   1:  PR[91,2] = PR[90,2] + 14.295;
   1:L PR[91] R[100]mm/sec CNT100;
   1:  PR[91,1] = PR[90,1] + 9.800;
   1:  PR[91,2] = PR[90,2] + 14.166;
   1:L PR[91] R[100]mm/sec CNT100;
   1:  PR[91,1] = PR[90,1] + 6.679;
   1:  PR[91,2] = PR[90,2] + 10.931;
   1:L PR[91] R[100]mm/sec CNT100;
   1:  PR[91,1] = PR[90,1] + 6.224;
   1:  PR[91,2] = PR[90,2] + 10.258;
   1:L PR[91] R[100]mm/sec CNT100;
   1:  PR[91,1] = PR[90,1] + 5.273;
   1:  PR[91,2] = PR[90,2] + 8.564;
   1:L PR[91] R[100]mm/sec CNT100;
   1:  PR[91,1] = PR[90,1] + 5.411;
   1:  PR[91,2] = PR[90,2] + 8.540;
   1:L PR[91] R[100]mm/sec CNT100;
   1:  PR[91,1] = PR[90,1] + 3.886;
   1:  PR[91,2] = PR[90,2] + 6.154;
   1:L PR[91] R[100]mm/sec CNT100;
   1:  PR[91,1] = PR[90,1] + 3.596;
   1:  PR[91,2] = PR[90,2] + 5.846;
   1:L PR[91] R[100]mm/sec CNT100;
   1:  PR[91,1] = PR[90,1] + 2.742;
   1:  PR[91,2] = PR[90,2] + 5.238;
   1:L PR[91] R[100]mm/sec CNT100;
   1:  PR[91,1] = PR[90,1] + 1.672;
   1:  PR[91,2] = PR[90,2] + 5.008;
   1:L PR[91] R[100]mm/sec CNT100;
   1:  PR[91,1] = PR[90,1] + -1.507;
   1:L PR[91] R[100]mm/sec CNT100;
   1:  PR[91] = PR[90];
   1:  PR[91,1] = PR[90,1] + -2.515;
   1:  PR[91,2] = PR[90,2] + 5.532;
   1:  PR[91,3] = PR[90,3] + 14.945;
   1:L PR[91] R[100]mm/sec CNT100;
   1:  PR[91,1] = PR[90,1] + -3.313;
   1:  PR[91,2] = PR[90,2] + 6.100;
   1:L PR[91] R[100]mm/sec CNT100;
   1:  PR[91,1] = PR[90,1] + -3.690;
   1:  PR[91,2] = PR[90,2] + 6.481;
   1:L PR[91] R[100]mm/sec CNT100;
   1:  PR[91,1] = PR[90,1] + -4.029;
   1:  PR[91,2] = PR[90,2] + 7.015;
   1:L PR[91] R[100]mm/sec CNT100;
   1:  PR[91,1] = PR[90,1] + -5.541;
   1:  PR[91,2] = PR[90,2] + 9.725;
   1:L PR[91] R[100]mm/sec CNT100;
   1:  PR[91,1] = PR[90,1] + -6.491;
   1:  PR[91,2] = PR[90,2] + 11.148;
   1:L PR[91] R[100]mm/sec CNT100;
   1:  PR[91,1] = PR[90,1] + -9.060;
   1:  PR[91,2] = PR[90,2] + 13.805;
   1:L PR[91] R[100]mm/sec CNT100;
   1:  PR[91,1] = PR[90,1] + -9.776;
   1:  PR[91,2] = PR[90,2] + 14.440;
   1:L PR[91] R[100]mm/sec CNT100;
   1:  PR[91,1] = PR[90,1] + -13.611;
   1:  PR[91,2] = PR[90,2] + 16.788;
   1:L PR[91] R[100]mm/sec CNT100;
   1:  PR[91,1] = PR[90,1] + -13.803;
   1:  PR[91,2] = PR[90,2] + 16.888;
   1:L PR[91] R[100]mm/sec CNT100;
   1:  PR[91,1] = PR[90,1] + -16.097;
   1:  PR[91,2] = PR[90,2] + 17.603;
   1:L PR[91] R[100]mm/sec CNT100;
   1:  PR[91,1] = PR[90,1] + -18.417;
   1:  PR[91,2] = PR[90,2] + 18.357;
   1:L PR[91] R[100]mm/sec CNT100;
   1:  PR[91,1] = PR[90,1] + -18.598;
   1:  PR[91,2] = PR[90,2] + 18.378;
   1:L PR[91] R[100]mm/sec CNT100;
   1:  PR[91,1] = PR[90,1] + -23.160;
   1:  PR[91,2] = PR[90,2] + 18.675;
   1:L PR[91] R[100]mm/sec CNT100;
   1:  PR[91,1] = PR[90,1] + -24.014;
   1:  PR[91,2] = PR[90,2] + 18.553;
   1:L PR[91] R[100]mm/sec CNT100;
   1:  PR[91,1] = PR[90,1] + -27.876;
   1:  PR[91,2] = PR[90,2] + 17.835;
   1:L PR[91] R[100]mm/sec CNT100;
   1:  PR[91,1] = PR[90,1] + -29.208;
   1:  PR[91,2] = PR[90,2] + 17.272;
   1:L PR[91] R[100]mm/sec CNT100;
   1:  PR[91,1] = PR[90,1] + -32.267;
   1:  PR[91,2] = PR[90,2] + 15.857;
   1:L PR[91] R[100]mm/sec CNT100;
   1:  PR[91,1] = PR[90,1] + -33.781;
   1:  PR[91,2] = PR[90,2] + 14.686;
   1:L PR[91] R[100]mm/sec CNT100;
   1:  PR[91,1] = PR[90,1] + -36.042;
   1:  PR[91,2] = PR[90,2] + 12.845;
   1:L PR[91] R[100]mm/sec CNT100;
   1:  PR[91,1] = PR[90,1] + -37.414;
   1:  PR[91,2] = PR[90,2] + 11.050;
   1:L PR[91] R[100]mm/sec CNT100;
   1:  PR[91,1] = PR[90,1] + -38.944;
   1:  PR[91,2] = PR[90,2] + 8.967;
   1:L PR[91] R[100]mm/sec CNT100;
   1:  PR[91,1] = PR[90,1] + -39.896;
   1:  PR[91,2] = PR[90,2] + 6.669;
   1:L PR[91] R[100]mm/sec CNT100;
   1:  PR[91,1] = PR[90,1] + -40.771;
   1:  PR[91,2] = PR[90,2] + 4.501;
   1:L PR[91] R[100]mm/sec CNT100;
   1:  PR[91,1] = PR[90,1] + -41.398;
   1:  PR[91,2] = PR[90,2] + -0.312;
   1:L PR[91] R[100]mm/sec CNT100;
   1:  PR[91,1] = PR[90,1] + -40.771;
   1:  PR[91,2] = PR[90,2] + -5.125;
   1:L PR[91] R[100]mm/sec CNT100;
   1:  PR[91,1] = PR[90,1] + -39.896;
   1:  PR[91,2] = PR[90,2] + -7.294;
   1:L PR[91] R[100]mm/sec CNT100;
   1:  PR[91,1] = PR[90,1] + -38.944;
   1:  PR[91,2] = PR[90,2] + -9.591;
   1:L PR[91] R[100]mm/sec CNT100;
   1:  PR[91,1] = PR[90,1] + -37.414;
   1:  PR[91,2] = PR[90,2] + -11.674;
   1:L PR[91] R[100]mm/sec CNT100;
   1:  PR[91,1] = PR[90,1] + -36.042;
   1:  PR[91,2] = PR[90,2] + -13.469;
   1:L PR[91] R[100]mm/sec CNT100;
   1:  PR[91,1] = PR[90,1] + -33.781;
   1:  PR[91,2] = PR[90,2] + -15.310;
   1:L PR[91] R[100]mm/sec CNT100;
   1:  PR[91,1] = PR[90,1] + -32.266;
   1:  PR[91,2] = PR[90,2] + -16.481;
   1:L PR[91] R[100]mm/sec CNT100;
   1:  PR[91,1] = PR[90,1] + -29.208;
   1:  PR[91,2] = PR[90,2] + -17.896;
   1:L PR[91] R[100]mm/sec CNT100;
   1:  PR[91,1] = PR[90,1] + -27.875;
   1:  PR[91,2] = PR[90,2] + -18.459;
   1:L PR[91] R[100]mm/sec CNT100;
   1:  PR[91,1] = PR[90,1] + -24.013;
   1:  PR[91,2] = PR[90,2] + -19.177;
   1:L PR[91] R[100]mm/sec CNT100;
   1:  PR[91,1] = PR[90,1] + -23.159;
   1:  PR[91,2] = PR[90,2] + -19.299;
   1:L PR[91] R[100]mm/sec CNT100;
   1:  PR[91,1] = PR[90,1] + -18.596;
   1:  PR[91,2] = PR[90,2] + -19.001;
   1:L PR[91] R[100]mm/sec CNT100;
   1:  PR[91,1] = PR[90,1] + -18.416;
   1:  PR[91,2] = PR[90,2] + -18.981;
   1:L PR[91] R[100]mm/sec CNT100;
   1:  PR[91,1] = PR[90,1] + -16.097;
   1:  PR[91,2] = PR[90,2] + -18.227;
   1:L PR[91] R[100]mm/sec CNT100;
   1:  PR[91,1] = PR[90,1] + -13.802;
   1:  PR[91,2] = PR[90,2] + -17.512;
   1:L PR[91] R[100]mm/sec CNT100;
   1:  PR[91,1] = PR[90,1] + -13.610;
   1:  PR[91,2] = PR[90,2] + -17.411;
   1:L PR[91] R[100]mm/sec CNT100;
   1:  PR[91,1] = PR[90,1] + -9.775;
   1:  PR[91,2] = PR[90,2] + -15.063;
   1:L PR[91] R[100]mm/sec CNT100;
   1:  PR[91,1] = PR[90,1] + -9.059;
   1:  PR[91,2] = PR[90,2] + -14.428;
   1:L PR[91] R[100]mm/sec CNT100;
   1:  PR[91,1] = PR[90,1] + -6.489;
   1:  PR[91,2] = PR[90,2] + -11.769;
   1:L PR[91] R[100]mm/sec CNT100;
   1:  PR[91,1] = PR[90,1] + -5.569;
   1:  PR[91,2] = PR[90,2] + -10.401;
   1:L PR[91] R[100]mm/sec CNT100;
   1:  PR[91,1] = PR[90,1] + -4.028;
   1:  PR[91,2] = PR[90,2] + -7.639;
   1:L PR[91] R[100]mm/sec CNT100;
   1:  PR[91,1] = PR[90,1] + -3.683;
   1:  PR[91,2] = PR[90,2] + -7.096;
   1:L PR[91] R[100]mm/sec CNT100;
   1:  PR[91,1] = PR[90,1] + -3.311;
   1:  PR[91,2] = PR[90,2] + -6.722;
   1:L PR[91] R[100]mm/sec CNT100;
   1:  PR[91,1] = PR[90,1] + -2.515;
   1:  PR[91,2] = PR[90,2] + -6.156;
   1:L PR[91] R[100]mm/sec CNT100;
   1:  PR[91,1] = PR[90,1] + -1.428;
   1:  PR[91,2] = PR[90,2] + -5.921;
   1:L PR[91] R[100]mm/sec CNT100;
   1:  PR[91,1] = PR[90,1] + 1.584;
   1:L PR[91] R[100]mm/sec CNT100;
   1:  PR[91,1] = PR[90,1] + 2.668;
   1:  PR[91,2] = PR[90,2] + -6.155;
   1:L PR[91] R[100]mm/sec CNT100;
   1:  PR[91,1] = PR[90,1] + 3.441;
   1:  PR[91,2] = PR[90,2] + -6.703;
   1:L PR[91] R[100]mm/sec CNT100;
   1:  PR[91,1] = PR[90,1] + 3.541;
   1:  PR[91,2] = PR[90,2] + -6.796;
   1:L PR[91] R[100]mm/sec CNT100;
   1:  PR[91,1] = PR[90,1] + 3.696;
   1:  PR[91,2] = PR[90,2] + -6.767;
   1:L PR[91] R[100]mm/sec CNT100;
   1:  PR[91,1] = PR[90,1] + 5.726;
   1:  PR[91,2] = PR[90,2] + -10.398;
   1:L PR[91] R[100]mm/sec CNT100;
   1:  PR[91,1] = PR[90,1] + 6.644;
   1:  PR[91,2] = PR[90,2] + -11.761;
   1:L PR[91] R[100]mm/sec CNT100;
   1:  PR[91,1] = PR[90,1] + 9.214;
   1:  PR[91,2] = PR[90,2] + -14.427;
   1:L PR[91] R[100]mm/sec CNT100;
   1:  PR[91,1] = PR[90,1] + 9.930;
   1:  PR[91,2] = PR[90,2] + -15.063;
   1:L PR[91] R[100]mm/sec CNT100;
   1:  PR[91,1] = PR[90,1] + 13.762;
   1:  PR[91,2] = PR[90,2] + -17.409;
   1:L PR[91] R[100]mm/sec CNT100;
   1:  PR[91,1] = PR[90,1] + 13.954;
   1:  PR[91,2] = PR[90,2] + -17.510;
   1:L PR[91] R[100]mm/sec CNT100;
   1:  PR[91,1] = PR[90,1] + 16.254;
   1:  PR[91,2] = PR[90,2] + -18.227;
   1:L PR[91] R[100]mm/sec CNT100;
   1:  PR[91,1] = PR[90,1] + 18.569;
   1:  PR[91,2] = PR[90,2] + -18.980;
   1:L PR[91] R[100]mm/sec CNT100;
   1:  PR[91,1] = PR[90,1] + 18.749;
   1:  PR[91,2] = PR[90,2] + -19.001;
   1:L PR[91] R[100]mm/sec CNT100;
   1:  PR[91,1] = PR[90,1] + 23.313;
   1:  PR[91,2] = PR[90,2] + -19.299;
   1:L PR[91] R[100]mm/sec CNT100;
   1:  PR[91,1] = PR[90,1] + 24.167;
   1:  PR[91,2] = PR[90,2] + -19.177;
   1:L PR[91] R[100]mm/sec CNT100;
   1:  PR[91,1] = PR[90,1] + 28.030;
   1:  PR[91,2] = PR[90,2] + -18.459;
   1:L PR[91] R[100]mm/sec CNT100;
   1:  PR[91,1] = PR[90,1] + 29.362;
   1:  PR[91,2] = PR[90,2] + -17.896;
   1:L PR[91] R[100]mm/sec CNT100;
   1:  PR[91,1] = PR[90,1] + 32.422;
   1:  PR[91,2] = PR[90,2] + -16.482;
   1:L PR[91] R[100]mm/sec CNT100;
   1:  PR[91,1] = PR[90,1] + 33.936;
   1:  PR[91,2] = PR[90,2] + -15.312;
   1:L PR[91] R[100]mm/sec CNT100;
   1:  PR[91,1] = PR[90,1] + 36.198;
   1:  PR[91,2] = PR[90,2] + -13.470;
   1:L PR[91] R[100]mm/sec CNT100;
   1:  PR[91,1] = PR[90,1] + 37.570;
   1:  PR[91,2] = PR[90,2] + -11.674;
   1:L PR[91] R[100]mm/sec CNT100;
   1:  PR[91,1] = PR[90,1] + 39.100;
   1:  PR[91,2] = PR[90,2] + -9.588;
   1:L PR[91] R[100]mm/sec CNT100;
   1:  PR[91,1] = PR[90,1] + 40.053;
   1:  PR[91,2] = PR[90,2] + -7.294;
   1:L PR[91] R[100]mm/sec CNT100;
   1:  PR[91,1] = PR[90,1] + 40.929;
   1:  PR[91,2] = PR[90,2] + -5.130;
   1:L PR[91] R[100]mm/sec CNT100;
   1:  PR[91,1] = PR[90,1] + 41.281;
   1:  PR[91,2] = PR[90,2] + -2.473;
   1:L PR[91] R[100]mm/sec CNT100;
   1:  PR[91,1] = PR[90,1] + 41.555;
   1:  PR[91,2] = PR[90,2] + -0.314;
   1:L PR[91] R[100]mm/sec CNT100;
   1:  PR[91,1] = PR[90,1] + 40.928;
   1:  PR[91,2] = PR[90,2] + 4.508;
   1:L PR[91] R[100]mm/sec CNT100;
   1:  PR[91,1] = PR[90,1] + 40.053;
   1:  PR[91,2] = PR[90,2] + 6.669;
   1:L PR[91] R[100]mm/sec CNT100;
   1:  PR[91,1] = PR[90,1] + 39.100;
   1:  PR[91,2] = PR[90,2] + 8.965;
   1:L PR[91] R[100]mm/sec CNT100;
   1:  PR[91,1] = PR[90,1] + 37.570;
   1:  PR[91,2] = PR[90,2] + 11.050;
   1:L PR[91] R[100]mm/sec CNT100;
   1:  PR[91,1] = PR[90,1] + 36.198;
   1:  PR[91,2] = PR[90,2] + 12.846;
   1:L PR[91] R[100]mm/sec CNT100;
   1:  PR[91,1] = PR[90,1] + 33.937;
   1:  PR[91,2] = PR[90,2] + 14.688;
   1:L PR[91] R[100]mm/sec CNT100;
   1:  PR[91,1] = PR[90,1] + 32.422;
   1:  PR[91,2] = PR[90,2] + 15.858;
   1:L PR[91] R[100]mm/sec CNT100;
   1:  PR[91,1] = PR[90,1] + 29.364;
   1:  PR[91,2] = PR[90,2] + 17.271;
   1:L PR[91] R[100]mm/sec CNT100;
   1:  PR[91,1] = PR[90,1] + 28.031;
   1:  PR[91,2] = PR[90,2] + 17.834;
   1:L PR[91] R[100]mm/sec CNT100;
   1:  PR[91,1] = PR[90,1] + 24.170;
   1:  PR[91,2] = PR[90,2] + 18.553;
   1:L PR[91] R[100]mm/sec CNT100;
   1:  PR[91,1] = PR[90,1] + 23.316;
   1:  PR[91,2] = PR[90,2] + 18.675;
   1:L PR[91] R[100]mm/sec CNT100;
   1:  PR[91,1] = PR[90,1] + 18.755;
   1:  PR[91,2] = PR[90,2] + 18.378;
   1:L PR[91] R[100]mm/sec CNT100;
   1:  PR[91,1] = PR[90,1] + 18.574;
   1:  PR[91,2] = PR[90,2] + 18.357;
   1:L PR[91] R[100]mm/sec CNT100;
   1:  PR[91,1] = PR[90,1] + 16.254;
   1:  PR[91,2] = PR[90,2] + 17.603;
   1:L PR[91] R[100]mm/sec CNT100;
   1:  PR[91,1] = PR[90,1] + 13.959;
   1:  PR[91,2] = PR[90,2] + 16.888;
   1:L PR[91] R[100]mm/sec CNT100;
   1:  PR[91,1] = PR[90,1] + 13.767;
   1:  PR[91,2] = PR[90,2] + 16.787;
   1:L PR[91] R[100]mm/sec CNT100;
   1:  PR[91,1] = PR[90,1] + 9.932;
   1:  PR[91,2] = PR[90,2] + 14.441;
   1:L PR[91] R[100]mm/sec CNT100;
   1:  PR[91,1] = PR[90,1] + 9.216;
   1:  PR[91,2] = PR[90,2] + 13.804;
   1:L PR[91] R[100]mm/sec CNT100;
   1:  PR[91,1] = PR[90,1] + 6.643;
   1:  PR[91,2] = PR[90,2] + 11.137;
   1:L PR[91] R[100]mm/sec CNT100;
   1:  PR[91,1] = PR[90,1] + 5.747;
   1:  PR[91,2] = PR[90,2] + 9.811;
   1:L PR[91] R[100]mm/sec CNT100;
   1:  PR[91,1] = PR[90,1] + 5.190;
   1:  PR[91,2] = PR[90,2] + 8.819;
   1:L PR[91] R[100]mm/sec CNT100;
   1:  PR[91,1] = PR[90,1] + 5.359;
   1:  PR[91,2] = PR[90,2] + 8.789;
   1:L PR[91] R[100]mm/sec CNT100;
   1:  PR[91,1] = PR[90,1] + 3.825;
   1:  PR[91,2] = PR[90,2] + 6.457;
   1:L PR[91] R[100]mm/sec CNT100;
   1:  PR[91,1] = PR[90,1] + 3.465;
   1:  PR[91,2] = PR[90,2] + 6.097;
   1:L PR[91] R[100]mm/sec CNT100;
   1:  PR[91,1] = PR[90,1] + 2.673;
   1:  PR[91,2] = PR[90,2] + 5.533;
   1:L PR[91] R[100]mm/sec CNT100;
   1:  PR[91,1] = PR[90,1] + 1.593;
   1:  PR[91,2] = PR[90,2] + 5.297;
   1:L PR[91] R[100]mm/sec CNT100;
   1:  PR[91,1] = PR[90,1] + -1.427;
   1:L PR[91] R[100]mm/sec CNT100;
   1:  PR[91] = PR[90];
   1:  PR[91,1] = PR[90,1] + -2.445;
   1:  PR[91,2] = PR[90,2] + 5.827;
   1:  PR[91,3] = PR[90,3] + 15.555;
   1:L PR[91] R[100]mm/sec CNT100;
   1:  PR[91,1] = PR[90,1] + -3.200;
   1:  PR[91,2] = PR[90,2] + 6.364;
   1:L PR[91] R[100]mm/sec CNT100;
   1:  PR[91,1] = PR[90,1] + -3.672;
   1:  PR[91,2] = PR[90,2] + 6.843;
   1:L PR[91] R[100]mm/sec CNT100;
   1:  PR[91,1] = PR[90,1] + -3.947;
   1:  PR[91,2] = PR[90,2] + 7.275;
   1:L PR[91] R[100]mm/sec CNT100;
   1:  PR[91,1] = PR[90,1] + -5.042;
   1:  PR[91,2] = PR[90,2] + 9.237;
   1:L PR[91] R[100]mm/sec CNT100;
   1:  PR[91,1] = PR[90,1] + -6.455;
   1:  PR[91,2] = PR[90,2] + 11.355;
   1:L PR[91] R[100]mm/sec CNT100;
   1:  PR[91,1] = PR[90,1] + -8.477;
   1:  PR[91,2] = PR[90,2] + 13.446;
   1:L PR[91] R[100]mm/sec CNT100;
   1:  PR[91,1] = PR[90,1] + -9.764;
   1:  PR[91,2] = PR[90,2] + 14.587;
   1:L PR[91] R[100]mm/sec CNT100;
   1:  PR[91,1] = PR[90,1] + -12.951;
   1:  PR[91,2] = PR[90,2] + 16.538;
   1:L PR[91] R[100]mm/sec CNT100;
   1:  PR[91,1] = PR[90,1] + -13.796;
   1:  PR[91,2] = PR[90,2] + 16.982;
   1:L PR[91] R[100]mm/sec CNT100;
   1:  PR[91,1] = PR[90,1] + -18.202;
   1:  PR[91,2] = PR[90,2] + 18.354;
   1:L PR[91] R[100]mm/sec CNT100;
   1:  PR[91,1] = PR[90,1] + -18.339;
   1:  PR[91,2] = PR[90,2] + 18.388;
   1:L PR[91] R[100]mm/sec CNT100;
   1:  PR[91,1] = PR[90,1] + -20.244;
   1:  PR[91,2] = PR[90,2] + 18.495;
   1:L PR[91] R[100]mm/sec CNT100;
   1:  PR[91,1] = PR[90,1] + -23.180;
   1:  PR[91,2] = PR[90,2] + 18.687;
   1:L PR[91] R[100]mm/sec CNT100;
   1:  PR[91,1] = PR[90,1] + -23.424;
   1:  PR[91,2] = PR[90,2] + 18.652;
   1:L PR[91] R[100]mm/sec CNT100;
   1:  PR[91,1] = PR[90,1] + -27.877;
   1:  PR[91,2] = PR[90,2] + 17.824;
   1:L PR[91] R[100]mm/sec CNT100;
   1:  PR[91,1] = PR[90,1] + -28.676;
   1:  PR[91,2] = PR[90,2] + 17.486;
   1:L PR[91] R[100]mm/sec CNT100;
   1:  PR[91,1] = PR[90,1] + -32.247;
   1:  PR[91,2] = PR[90,2] + 15.834;
   1:L PR[91] R[100]mm/sec CNT100;
   1:  PR[91,1] = PR[90,1] + -33.331;
   1:  PR[91,2] = PR[90,2] + 14.997;
   1:L PR[91] R[100]mm/sec CNT100;
   1:  PR[91,1] = PR[90,1] + -36.004;
   1:  PR[91,2] = PR[90,2] + 12.821;
   1:L PR[91] R[100]mm/sec CNT100;
   1:  PR[91,1] = PR[90,1] + -37.062;
   1:  PR[91,2] = PR[90,2] + 11.436;
   1:L PR[91] R[100]mm/sec CNT100;
   1:  PR[91,1] = PR[90,1] + -38.891;
   1:  PR[91,2] = PR[90,2] + 8.946;
   1:L PR[91] R[100]mm/sec CNT100;
   1:  PR[91,1] = PR[90,1] + -39.654;
   1:  PR[91,2] = PR[90,2] + 7.105;
   1:L PR[91] R[100]mm/sec CNT100;
   1:  PR[91,1] = PR[90,1] + -40.709;
   1:  PR[91,2] = PR[90,2] + 4.492;
   1:L PR[91] R[100]mm/sec CNT100;
   1:  PR[91,1] = PR[90,1] + -41.332;
   1:  PR[91,2] = PR[90,2] + -0.312;
   1:L PR[91] R[100]mm/sec CNT100;
   1:  PR[91,1] = PR[90,1] + -40.709;
   1:  PR[91,2] = PR[90,2] + -5.116;
   1:L PR[91] R[100]mm/sec CNT100;
   1:  PR[91,1] = PR[90,1] + -39.653;
   1:  PR[91,2] = PR[90,2] + -7.730;
   1:L PR[91] R[100]mm/sec CNT100;
   1:  PR[91,1] = PR[90,1] + -38.891;
   1:  PR[91,2] = PR[90,2] + -9.570;
   1:L PR[91] R[100]mm/sec CNT100;
   1:  PR[91,1] = PR[90,1] + -37.062;
   1:  PR[91,2] = PR[90,2] + -12.060;
   1:L PR[91] R[100]mm/sec CNT100;
   1:  PR[91,1] = PR[90,1] + -36.003;
   1:  PR[91,2] = PR[90,2] + -13.445;
   1:L PR[91] R[100]mm/sec CNT100;
   1:  PR[91,1] = PR[90,1] + -33.330;
   1:  PR[91,2] = PR[90,2] + -15.621;
   1:L PR[91] R[100]mm/sec CNT100;
   1:  PR[91,1] = PR[90,1] + -32.247;
   1:  PR[91,2] = PR[90,2] + -16.459;
   1:L PR[91] R[100]mm/sec CNT100;
   1:  PR[91,1] = PR[90,1] + -28.676;
   1:  PR[91,2] = PR[90,2] + -18.111;
   1:L PR[91] R[100]mm/sec CNT100;
   1:  PR[91,1] = PR[90,1] + -27.876;
   1:  PR[91,2] = PR[90,2] + -18.449;
   1:L PR[91] R[100]mm/sec CNT100;
   1:  PR[91,1] = PR[90,1] + -23.422;
   1:  PR[91,2] = PR[90,2] + -19.276;
   1:L PR[91] R[100]mm/sec CNT100;
   1:  PR[91,1] = PR[90,1] + -23.180;
   1:  PR[91,2] = PR[90,2] + -19.311;
   1:L PR[91] R[100]mm/sec CNT100;
   1:  PR[91,1] = PR[90,1] + -20.244;
   1:  PR[91,2] = PR[90,2] + -19.119;
   1:L PR[91] R[100]mm/sec CNT100;
   1:  PR[91,1] = PR[90,1] + -18.338;
   1:  PR[91,2] = PR[90,2] + -19.012;
   1:L PR[91] R[100]mm/sec CNT100;
   1:  PR[91,1] = PR[90,1] + -18.201;
   1:  PR[91,2] = PR[90,2] + -18.978;
   1:L PR[91] R[100]mm/sec CNT100;
   1:  PR[91,1] = PR[90,1] + -13.795;
   1:  PR[91,2] = PR[90,2] + -17.606;
   1:L PR[91] R[100]mm/sec CNT100;
   1:  PR[91,1] = PR[90,1] + -12.950;
   1:  PR[91,2] = PR[90,2] + -17.162;
   1:L PR[91] R[100]mm/sec CNT100;
   1:  PR[91,1] = PR[90,1] + -9.763;
   1:  PR[91,2] = PR[90,2] + -15.210;
   1:L PR[91] R[100]mm/sec CNT100;
   1:  PR[91,1] = PR[90,1] + -8.476;
   1:  PR[91,2] = PR[90,2] + -14.069;
   1:L PR[91] R[100]mm/sec CNT100;
   1:  PR[91,1] = PR[90,1] + -6.453;
   1:  PR[91,2] = PR[90,2] + -11.977;
   1:L PR[91] R[100]mm/sec CNT100;
   1:  PR[91,1] = PR[90,1] + -5.082;
   1:  PR[91,2] = PR[90,2] + -9.937;
   1:L PR[91] R[100]mm/sec CNT100;
   1:  PR[91,1] = PR[90,1] + -3.945;
   1:  PR[91,2] = PR[90,2] + -7.899;
   1:L PR[91] R[100]mm/sec CNT100;
   1:  PR[91,1] = PR[90,1] + -3.663;
   1:  PR[91,2] = PR[90,2] + -7.454;
   1:L PR[91] R[100]mm/sec CNT100;
   1:  PR[91,1] = PR[90,1] + -3.197;
   1:  PR[91,2] = PR[90,2] + -6.986;
   1:L PR[91] R[100]mm/sec CNT100;
   1:  PR[91,1] = PR[90,1] + -2.445;
   1:  PR[91,2] = PR[90,2] + -6.451;
   1:L PR[91] R[100]mm/sec CNT100;
   1:  PR[91,1] = PR[90,1] + -1.349;
   1:  PR[91,2] = PR[90,2] + -6.209;
   1:L PR[91] R[100]mm/sec CNT100;
   1:  PR[91,1] = PR[90,1] + 1.505;
   1:L PR[91] R[100]mm/sec CNT100;
   1:  PR[91,1] = PR[90,1] + 2.599;
   1:  PR[91,2] = PR[90,2] + -6.450;
   1:L PR[91] R[100]mm/sec CNT100;
   1:  PR[91,1] = PR[90,1] + 3.328;
   1:  PR[91,2] = PR[90,2] + -6.967;
   1:L PR[91] R[100]mm/sec CNT100;
   1:  PR[91,1] = PR[90,1] + 3.430;
   1:  PR[91,2] = PR[90,2] + -7.062;
   1:L PR[91] R[100]mm/sec CNT100;
   1:  PR[91,1] = PR[90,1] + 3.614;
   1:  PR[91,2] = PR[90,2] + -7.027;
   1:L PR[91] R[100]mm/sec CNT100;
   1:  PR[91,1] = PR[90,1] + 5.241;
   1:  PR[91,2] = PR[90,2] + -9.937;
   1:L PR[91] R[100]mm/sec CNT100;
   1:  PR[91,1] = PR[90,1] + 6.608;
   1:  PR[91,2] = PR[90,2] + -11.969;
   1:L PR[91] R[100]mm/sec CNT100;
   1:  PR[91,1] = PR[90,1] + 8.632;
   1:  PR[91,2] = PR[90,2] + -14.068;
   1:L PR[91] R[100]mm/sec CNT100;
   1:  PR[91,1] = PR[90,1] + 9.918;
   1:  PR[91,2] = PR[90,2] + -15.211;
   1:L PR[91] R[100]mm/sec CNT100;
   1:  PR[91,1] = PR[90,1] + 13.103;
   1:  PR[91,2] = PR[90,2] + -17.160;
   1:L PR[91] R[100]mm/sec CNT100;
   1:  PR[91,1] = PR[90,1] + 13.948;
   1:  PR[91,2] = PR[90,2] + -17.604;
   1:L PR[91] R[100]mm/sec CNT100;
   1:  PR[91,1] = PR[90,1] + 18.354;
   1:  PR[91,2] = PR[90,2] + -18.977;
   1:L PR[91] R[100]mm/sec CNT100;
   1:  PR[91,1] = PR[90,1] + 18.492;
   1:  PR[91,2] = PR[90,2] + -19.011;
   1:L PR[91] R[100]mm/sec CNT100;
   1:  PR[91,1] = PR[90,1] + 20.401;
   1:  PR[91,2] = PR[90,2] + -19.119;
   1:L PR[91] R[100]mm/sec CNT100;
   1:  PR[91,1] = PR[90,1] + 23.334;
   1:  PR[91,2] = PR[90,2] + -19.311;
   1:L PR[91] R[100]mm/sec CNT100;
   1:  PR[91,1] = PR[90,1] + 23.576;
   1:  PR[91,2] = PR[90,2] + -19.276;
   1:L PR[91] R[100]mm/sec CNT100;
   1:  PR[91,1] = PR[90,1] + 28.031;
   1:  PR[91,2] = PR[90,2] + -18.448;
   1:L PR[91] R[100]mm/sec CNT100;
   1:  PR[91,1] = PR[90,1] + 28.830;
   1:  PR[91,2] = PR[90,2] + -18.110;
   1:L PR[91] R[100]mm/sec CNT100;
   1:  PR[91,1] = PR[90,1] + 32.402;
   1:  PR[91,2] = PR[90,2] + -16.460;
   1:L PR[91] R[100]mm/sec CNT100;
   1:  PR[91,1] = PR[90,1] + 33.485;
   1:  PR[91,2] = PR[90,2] + -15.623;
   1:L PR[91] R[100]mm/sec CNT100;
   1:  PR[91,1] = PR[90,1] + 36.159;
   1:  PR[91,2] = PR[90,2] + -13.446;
   1:L PR[91] R[100]mm/sec CNT100;
   1:  PR[91,1] = PR[90,1] + 37.217;
   1:  PR[91,2] = PR[90,2] + -12.061;
   1:L PR[91] R[100]mm/sec CNT100;
   1:  PR[91,1] = PR[90,1] + 39.047;
   1:  PR[91,2] = PR[90,2] + -9.567;
   1:L PR[91] R[100]mm/sec CNT100;
   1:  PR[91,1] = PR[90,1] + 39.810;
   1:  PR[91,2] = PR[90,2] + -7.728;
   1:L PR[91] R[100]mm/sec CNT100;
   1:  PR[91,1] = PR[90,1] + 40.866;
   1:  PR[91,2] = PR[90,2] + -5.121;
   1:L PR[91] R[100]mm/sec CNT100;
   1:  PR[91,1] = PR[90,1] + 41.154;
   1:  PR[91,2] = PR[90,2] + -2.953;
   1:L PR[91] R[100]mm/sec CNT100;
   1:  PR[91,1] = PR[90,1] + 41.489;
   1:  PR[91,2] = PR[90,2] + -0.314;
   1:L PR[91] R[100]mm/sec CNT100;
   1:  PR[91,1] = PR[90,1] + 40.865;
   1:  PR[91,2] = PR[90,2] + 4.499;
   1:L PR[91] R[100]mm/sec CNT100;
   1:  PR[91,1] = PR[90,1] + 39.811;
   1:  PR[91,2] = PR[90,2] + 7.103;
   1:L PR[91] R[100]mm/sec CNT100;
   1:  PR[91,1] = PR[90,1] + 39.047;
   1:  PR[91,2] = PR[90,2] + 8.943;
   1:L PR[91] R[100]mm/sec CNT100;
   1:  PR[91,1] = PR[90,1] + 37.218;
   1:  PR[91,2] = PR[90,2] + 11.436;
   1:L PR[91] R[100]mm/sec CNT100;
   1:  PR[91,1] = PR[90,1] + 36.159;
   1:  PR[91,2] = PR[90,2] + 12.821;
   1:L PR[91] R[100]mm/sec CNT100;
   1:  PR[91,1] = PR[90,1] + 33.487;
   1:  PR[91,2] = PR[90,2] + 14.999;
   1:L PR[91] R[100]mm/sec CNT100;
   1:  PR[91,1] = PR[90,1] + 32.403;
   1:  PR[91,2] = PR[90,2] + 15.836;
   1:L PR[91] R[100]mm/sec CNT100;
   1:  PR[91,1] = PR[90,1] + 28.833;
   1:  PR[91,2] = PR[90,2] + 17.486;
   1:L PR[91] R[100]mm/sec CNT100;
   1:  PR[91,1] = PR[90,1] + 28.032;
   1:  PR[91,2] = PR[90,2] + 17.824;
   1:L PR[91] R[100]mm/sec CNT100;
   1:  PR[91,1] = PR[90,1] + 23.580;
   1:  PR[91,2] = PR[90,2] + 18.652;
   1:L PR[91] R[100]mm/sec CNT100;
   1:  PR[91,1] = PR[90,1] + 23.337;
   1:  PR[91,2] = PR[90,2] + 18.687;
   1:L PR[91] R[100]mm/sec CNT100;
   1:  PR[91,1] = PR[90,1] + 20.401;
   1:  PR[91,2] = PR[90,2] + 18.495;
   1:L PR[91] R[100]mm/sec CNT100;
   1:  PR[91,1] = PR[90,1] + 18.497;
   1:  PR[91,2] = PR[90,2] + 18.388;
   1:L PR[91] R[100]mm/sec CNT100;
   1:  PR[91,1] = PR[90,1] + 18.359;
   1:  PR[91,2] = PR[90,2] + 18.354;
   1:L PR[91] R[100]mm/sec CNT100;
   1:  PR[91,1] = PR[90,1] + 13.951;
   1:  PR[91,2] = PR[90,2] + 16.981;
   1:L PR[91] R[100]mm/sec CNT100;
   1:  PR[91,1] = PR[90,1] + 13.105;
   1:  PR[91,2] = PR[90,2] + 16.537;
   1:L PR[91] R[100]mm/sec CNT100;
   1:  PR[91,1] = PR[90,1] + 9.918;
   1:  PR[91,2] = PR[90,2] + 14.588;
   1:L PR[91] R[100]mm/sec CNT100;
   1:  PR[91,1] = PR[90,1] + 8.631;
   1:  PR[91,2] = PR[90,2] + 13.442;
   1:L PR[91] R[100]mm/sec CNT100;
   1:  PR[91,1] = PR[90,1] + 6.606;
   1:  PR[91,2] = PR[90,2] + 11.343;
   1:L PR[91] R[100]mm/sec CNT100;
   1:  PR[91,1] = PR[90,1] + 5.270;
   1:  PR[91,2] = PR[90,2] + 9.365;
   1:L PR[91] R[100]mm/sec CNT100;
   1:  PR[91,1] = PR[90,1] + 5.107;
   1:  PR[91,2] = PR[90,2] + 9.076;
   1:L PR[91] R[100]mm/sec CNT100;
   1:  PR[91,1] = PR[90,1] + 5.248;
   1:  PR[91,2] = PR[90,2] + 9.051;
   1:L PR[91] R[100]mm/sec CNT100;
   1:  PR[91,1] = PR[90,1] + 3.904;
   1:  PR[91,2] = PR[90,2] + 6.949;
   1:L PR[91] R[100]mm/sec CNT100;
   1:  PR[91,1] = PR[90,1] + 3.586;
   1:  PR[91,2] = PR[90,2] + 6.582;
   1:L PR[91] R[100]mm/sec CNT100;
   1:  PR[91,1] = PR[90,1] + 3.331;
   1:  PR[91,2] = PR[90,2] + 6.346;
   1:L PR[91] R[100]mm/sec CNT100;
   1:  PR[91,1] = PR[90,1] + 2.603;
   1:  PR[91,2] = PR[90,2] + 5.828;
   1:L PR[91] R[100]mm/sec CNT100;
   1:  PR[91,1] = PR[90,1] + 1.513;
   1:  PR[91,2] = PR[90,2] + 5.585;
   1:L PR[91] R[100]mm/sec CNT100;
   1:  PR[91,1] = PR[90,1] + -1.348;
   1:L PR[91] R[100]mm/sec CNT100;
   1:  PR[91] = PR[90];
   1:  PR[91,1] = PR[90,1] + -2.375;
   1:  PR[91,2] = PR[90,2] + 6.122;
   1:  PR[91,3] = PR[90,3] + 16.165;
   1:L PR[91] R[100]mm/sec CNT100;
   1:  PR[91,1] = PR[90,1] + -3.061;
   1:  PR[91,2] = PR[90,2] + 6.611;
   1:L PR[91] R[100]mm/sec CNT100;
   1:  PR[91,1] = PR[90,1] + -3.346;
   1:  PR[91,2] = PR[90,2] + 6.876;
   1:L PR[91] R[100]mm/sec CNT100;
   1:  PR[91,1] = PR[90,1] + -3.693;
   1:  PR[91,2] = PR[90,2] + 7.253;
   1:L PR[91] R[100]mm/sec CNT100;
   1:  PR[91,1] = PR[90,1] + -4.539;
   1:  PR[91,2] = PR[90,2] + 8.744;
   1:L PR[91] R[100]mm/sec CNT100;
   1:  PR[91,1] = PR[90,1] + -6.420;
   1:  PR[91,2] = PR[90,2] + 11.562;
   1:L PR[91] R[100]mm/sec CNT100;
   1:  PR[91,1] = PR[90,1] + -7.895;
   1:  PR[91,2] = PR[90,2] + 13.088;
   1:L PR[91] R[100]mm/sec CNT100;
   1:  PR[91,1] = PR[90,1] + -9.752;
   1:  PR[91,2] = PR[90,2] + 14.734;
   1:L PR[91] R[100]mm/sec CNT100;
   1:  PR[91,1] = PR[90,1] + -12.291;
   1:  PR[91,2] = PR[90,2] + 16.289;
   1:L PR[91] R[100]mm/sec CNT100;
   1:  PR[91,1] = PR[90,1] + -13.790;
   1:  PR[91,2] = PR[90,2] + 17.076;
   1:L PR[91] R[100]mm/sec CNT100;
   1:  PR[91,1] = PR[90,1] + -17.504;
   1:  PR[91,2] = PR[90,2] + 18.232;
   1:L PR[91] R[100]mm/sec CNT100;
   1:  PR[91,1] = PR[90,1] + -18.325;
   1:  PR[91,2] = PR[90,2] + 18.438;
   1:L PR[91] R[100]mm/sec CNT100;
   1:  PR[91,1] = PR[90,1] + -23.080;
   1:  PR[91,2] = PR[90,2] + 18.705;
   1:L PR[91] R[100]mm/sec CNT100;
   1:  PR[91,1] = PR[90,1] + -23.114;
   1:  PR[91,2] = PR[90,2] + 18.706;
   1:L PR[91] R[100]mm/sec CNT100;
   1:  PR[91,1] = PR[90,1] + -27.877;
   1:  PR[91,2] = PR[90,2] + 17.814;
   1:L PR[91] R[100]mm/sec CNT100;
   1:  PR[91,1] = PR[90,1] + -28.144;
   1:  PR[91,2] = PR[90,2] + 17.701;
   1:L PR[91] R[100]mm/sec CNT100;
   1:  PR[91,1] = PR[90,1] + -32.227;
   1:  PR[91,2] = PR[90,2] + 15.812;
   1:L PR[91] R[100]mm/sec CNT100;
   1:  PR[91,1] = PR[90,1] + -32.880;
   1:  PR[91,2] = PR[90,2] + 15.308;
   1:L PR[91] R[100]mm/sec CNT100;
   1:  PR[91,1] = PR[90,1] + -35.965;
   1:  PR[91,2] = PR[90,2] + 12.796;
   1:L PR[91] R[100]mm/sec CNT100;
   1:  PR[91,1] = PR[90,1] + -36.709;
   1:  PR[91,2] = PR[90,2] + 11.823;
   1:L PR[91] R[100]mm/sec CNT100;
   1:  PR[91,1] = PR[90,1] + -38.838;
   1:  PR[91,2] = PR[90,2] + 8.924;
   1:L PR[91] R[100]mm/sec CNT100;
   1:  PR[91,1] = PR[90,1] + -39.411;
   1:  PR[91,2] = PR[90,2] + 7.541;
   1:L PR[91] R[100]mm/sec CNT100;
   1:  PR[91,1] = PR[90,1] + -40.646;
   1:  PR[91,2] = PR[90,2] + 4.482;
   1:L PR[91] R[100]mm/sec CNT100;
   1:  PR[91,1] = PR[90,1] + -41.266;
   1:  PR[91,2] = PR[90,2] + -0.312;
   1:L PR[91] R[100]mm/sec CNT100;
   1:  PR[91,1] = PR[90,1] + -40.646;
   1:  PR[91,2] = PR[90,2] + -5.106;
   1:L PR[91] R[100]mm/sec CNT100;
   1:  PR[91,1] = PR[90,1] + -39.411;
   1:  PR[91,2] = PR[90,2] + -8.165;
   1:L PR[91] R[100]mm/sec CNT100;
   1:  PR[91,1] = PR[90,1] + -38.838;
   1:  PR[91,2] = PR[90,2] + -9.549;
   1:L PR[91] R[100]mm/sec CNT100;
   1:  PR[91,1] = PR[90,1] + -36.709;
   1:  PR[91,2] = PR[90,2] + -12.447;
   1:L PR[91] R[100]mm/sec CNT100;
   1:  PR[91,1] = PR[90,1] + -35.965;
   1:  PR[91,2] = PR[90,2] + -13.421;
   1:L PR[91] R[100]mm/sec CNT100;
   1:  PR[91,1] = PR[90,1] + -32.880;
   1:  PR[91,2] = PR[90,2] + -15.932;
   1:L PR[91] R[100]mm/sec CNT100;
   1:  PR[91,1] = PR[90,1] + -32.227;
   1:  PR[91,2] = PR[90,2] + -16.436;
   1:L PR[91] R[100]mm/sec CNT100;
   1:  PR[91,1] = PR[90,1] + -28.143;
   1:  PR[91,2] = PR[90,2] + -18.326;
   1:L PR[91] R[100]mm/sec CNT100;
   1:  PR[91,1] = PR[90,1] + -27.876;
   1:  PR[91,2] = PR[90,2] + -18.438;
   1:L PR[91] R[100]mm/sec CNT100;
   1:  PR[91,1] = PR[90,1] + -23.146;
   1:  PR[91,2] = PR[90,2] + -19.324;
   1:L PR[91] R[100]mm/sec CNT100;
   1:  PR[91,1] = PR[90,1] + -18.323;
   1:  PR[91,2] = PR[90,2] + -19.061;
   1:L PR[91] R[100]mm/sec CNT100;
   1:  PR[91,1] = PR[90,1] + -17.503;
   1:  PR[91,2] = PR[90,2] + -18.856;
   1:L PR[91] R[100]mm/sec CNT100;
   1:  PR[91,1] = PR[90,1] + -13.789;
   1:  PR[91,2] = PR[90,2] + -17.700;
   1:L PR[91] R[100]mm/sec CNT100;
   1:  PR[91,1] = PR[90,1] + -12.290;
   1:  PR[91,2] = PR[90,2] + -16.912;
   1:L PR[91] R[100]mm/sec CNT100;
   1:  PR[91,1] = PR[90,1] + -9.751;
   1:  PR[91,2] = PR[90,2] + -15.357;
   1:L PR[91] R[100]mm/sec CNT100;
   1:  PR[91,1] = PR[90,1] + -7.894;
   1:  PR[91,2] = PR[90,2] + -13.711;
   1:L PR[91] R[100]mm/sec CNT100;
   1:  PR[91,1] = PR[90,1] + -6.418;
   1:  PR[91,2] = PR[90,2] + -12.184;
   1:L PR[91] R[100]mm/sec CNT100;
   1:  PR[91,1] = PR[90,1] + -4.596;
   1:  PR[91,2] = PR[90,2] + -9.472;
   1:L PR[91] R[100]mm/sec CNT100;
   1:  PR[91,1] = PR[90,1] + -3.863;
   1:  PR[91,2] = PR[90,2] + -8.159;
   1:L PR[91] R[100]mm/sec CNT100;
   1:  PR[91,1] = PR[90,1] + -3.643;
   1:  PR[91,2] = PR[90,2] + -7.812;
   1:L PR[91] R[100]mm/sec CNT100;
   1:  PR[91,1] = PR[90,1] + -3.084;
   1:  PR[91,2] = PR[90,2] + -7.250;
   1:L PR[91] R[100]mm/sec CNT100;
   1:  PR[91,1] = PR[90,1] + -2.374;
   1:  PR[91,2] = PR[90,2] + -6.746;
   1:L PR[91] R[100]mm/sec CNT100;
   1:  PR[91,1] = PR[90,1] + -1.269;
   1:  PR[91,2] = PR[90,2] + -6.498;
   1:L PR[91] R[100]mm/sec CNT100;
   1:  PR[91,1] = PR[90,1] + 1.427;
   1:L PR[91] R[100]mm/sec CNT100;
   1:  PR[91,1] = PR[90,1] + 2.530;
   1:  PR[91,2] = PR[90,2] + -6.745;
   1:L PR[91] R[100]mm/sec CNT100;
   1:  PR[91,1] = PR[90,1] + 3.215;
   1:  PR[91,2] = PR[90,2] + -7.231;
   1:L PR[91] R[100]mm/sec CNT100;
   1:  PR[91,1] = PR[90,1] + 3.318;
   1:  PR[91,2] = PR[90,2] + -7.327;
   1:L PR[91] R[100]mm/sec CNT100;
   1:  PR[91,1] = PR[90,1] + 3.532;
   1:  PR[91,2] = PR[90,2] + -7.286;
   1:L PR[91] R[100]mm/sec CNT100;
   1:  PR[91,1] = PR[90,1] + 4.756;
   1:  PR[91,2] = PR[90,2] + -9.476;
   1:L PR[91] R[100]mm/sec CNT100;
   1:  PR[91,1] = PR[90,1] + 6.573;
   1:  PR[91,2] = PR[90,2] + -12.177;
   1:L PR[91] R[100]mm/sec CNT100;
   1:  PR[91,1] = PR[90,1] + 8.050;
   1:  PR[91,2] = PR[90,2] + -13.709;
   1:L PR[91] R[100]mm/sec CNT100;
   1:  PR[91,1] = PR[90,1] + 9.906;
   1:  PR[91,2] = PR[90,2] + -15.359;
   1:L PR[91] R[100]mm/sec CNT100;
   1:  PR[91,1] = PR[90,1] + 12.444;
   1:  PR[91,2] = PR[90,2] + -16.912;
   1:L PR[91] R[100]mm/sec CNT100;
   1:  PR[91,1] = PR[90,1] + 13.943;
   1:  PR[91,2] = PR[90,2] + -17.698;
   1:L PR[91] R[100]mm/sec CNT100;
   1:  PR[91,1] = PR[90,1] + 17.656;
   1:  PR[91,2] = PR[90,2] + -18.855;
   1:L PR[91] R[100]mm/sec CNT100;
   1:  PR[91,1] = PR[90,1] + 18.478;
   1:  PR[91,2] = PR[90,2] + -19.061;
   1:L PR[91] R[100]mm/sec CNT100;
   1:  PR[91,1] = PR[90,1] + 23.232;
   1:  PR[91,2] = PR[90,2] + -19.330;
   1:L PR[91] R[100]mm/sec CNT100;
   1:  PR[91,1] = PR[90,1] + 23.266;
   1:L PR[91] R[100]mm/sec CNT100;
   1:  PR[91,1] = PR[90,1] + 28.031;
   1:  PR[91,2] = PR[90,2] + -18.438;
   1:L PR[91] R[100]mm/sec CNT100;
   1:  PR[91,1] = PR[90,1] + 28.298;
   1:  PR[91,2] = PR[90,2] + -18.325;
   1:L PR[91] R[100]mm/sec CNT100;
   1:  PR[91,1] = PR[90,1] + 32.382;
   1:  PR[91,2] = PR[90,2] + -16.439;
   1:L PR[91] R[100]mm/sec CNT100;
   1:  PR[91,1] = PR[90,1] + 33.035;
   1:  PR[91,2] = PR[90,2] + -15.934;
   1:L PR[91] R[100]mm/sec CNT100;
   1:  PR[91,1] = PR[90,1] + 36.121;
   1:  PR[91,2] = PR[90,2] + -13.421;
   1:L PR[91] R[100]mm/sec CNT100;
   1:  PR[91,1] = PR[90,1] + 36.865;
   1:  PR[91,2] = PR[90,2] + -12.447;
   1:L PR[91] R[100]mm/sec CNT100;
   1:  PR[91,1] = PR[90,1] + 38.992;
   1:  PR[91,2] = PR[90,2] + -9.549;
   1:L PR[91] R[100]mm/sec CNT100;
   1:  PR[91,1] = PR[90,1] + 40.804;
   1:  PR[91,2] = PR[90,2] + -5.110;
   1:L PR[91] R[100]mm/sec CNT100;
   1:  PR[91,1] = PR[90,1] + 41.026;
   1:  PR[91,2] = PR[90,2] + -3.432;
   1:L PR[91] R[100]mm/sec CNT100;
   1:  PR[91,1] = PR[90,1] + 41.423;
   1:  PR[91,2] = PR[90,2] + -0.313;
   1:L PR[91] R[100]mm/sec CNT100;
   1:  PR[91,1] = PR[90,1] + 40.803;
   1:  PR[91,2] = PR[90,2] + 4.488;
   1:L PR[91] R[100]mm/sec CNT100;
   1:  PR[91,1] = PR[90,1] + 38.992;
   1:  PR[91,2] = PR[90,2] + 8.925;
   1:L PR[91] R[100]mm/sec CNT100;
   1:  PR[91,1] = PR[90,1] + 36.866;
   1:  PR[91,2] = PR[90,2] + 11.822;
   1:L PR[91] R[100]mm/sec CNT100;
   1:  PR[91,1] = PR[90,1] + 36.121;
   1:  PR[91,2] = PR[90,2] + 12.797;
   1:L PR[91] R[100]mm/sec CNT100;
   1:  PR[91,1] = PR[90,1] + 33.036;
   1:  PR[91,2] = PR[90,2] + 15.309;
   1:L PR[91] R[100]mm/sec CNT100;
   1:  PR[91,1] = PR[90,1] + 32.384;
   1:  PR[91,2] = PR[90,2] + 15.814;
   1:L PR[91] R[100]mm/sec CNT100;
   1:  PR[91,1] = PR[90,1] + 28.301;
   1:  PR[91,2] = PR[90,2] + 17.700;
   1:L PR[91] R[100]mm/sec CNT100;
   1:  PR[91,1] = PR[90,1] + 28.033;
   1:  PR[91,2] = PR[90,2] + 17.813;
   1:L PR[91] R[100]mm/sec CNT100;
   1:  PR[91,1] = PR[90,1] + 23.271;
   1:  PR[91,2] = PR[90,2] + 18.706;
   1:L PR[91] R[100]mm/sec CNT100;
   1:  PR[91,1] = PR[90,1] + 23.237;
   1:L PR[91] R[100]mm/sec CNT100;
   1:  PR[91,1] = PR[90,1] + 18.481;
   1:  PR[91,2] = PR[90,2] + 18.438;
   1:L PR[91] R[100]mm/sec CNT100;
   1:  PR[91,1] = PR[90,1] + 17.659;
   1:  PR[91,2] = PR[90,2] + 18.231;
   1:L PR[91] R[100]mm/sec CNT100;
   1:  PR[91,1] = PR[90,1] + 13.943;
   1:  PR[91,2] = PR[90,2] + 17.074;
   1:L PR[91] R[100]mm/sec CNT100;
   1:  PR[91,1] = PR[90,1] + 12.443;
   1:  PR[91,2] = PR[90,2] + 16.286;
   1:L PR[91] R[100]mm/sec CNT100;
   1:  PR[91,1] = PR[90,1] + 9.905;
   1:  PR[91,2] = PR[90,2] + 14.734;
   1:L PR[91] R[100]mm/sec CNT100;
   1:  PR[91,1] = PR[90,1] + 8.047;
   1:  PR[91,2] = PR[90,2] + 13.080;
   1:L PR[91] R[100]mm/sec CNT100;
   1:  PR[91,1] = PR[90,1] + 6.569;
   1:  PR[91,2] = PR[90,2] + 11.548;
   1:L PR[91] R[100]mm/sec CNT100;
   1:  PR[91,1] = PR[90,1] + 5.069;
   1:  PR[91,2] = PR[90,2] + 9.328;
   1:L PR[91] R[100]mm/sec CNT100;
   1:  PR[91,1] = PR[90,1] + 5.169;
   1:  PR[91,2] = PR[90,2] + 9.311;
   1:L PR[91] R[100]mm/sec CNT100;
   1:  PR[91,1] = PR[90,1] + 3.905;
   1:  PR[91,2] = PR[90,2] + 7.334;
   1:L PR[91] R[100]mm/sec CNT100;
   1:  PR[91,1] = PR[90,1] + 3.518;
   1:  PR[91,2] = PR[90,2] + 6.888;
   1:L PR[91] R[100]mm/sec CNT100;
   1:  PR[91,1] = PR[90,1] + 3.218;
   1:  PR[91,2] = PR[90,2] + 6.610;
   1:L PR[91] R[100]mm/sec CNT100;
   1:  PR[91,1] = PR[90,1] + 2.533;
   1:  PR[91,2] = PR[90,2] + 6.123;
   1:L PR[91] R[100]mm/sec CNT100;
   1:  PR[91,1] = PR[90,1] + 1.434;
   1:  PR[91,2] = PR[90,2] + 5.874;
   1:L PR[91] R[100]mm/sec CNT100;
   1:  PR[91,1] = PR[90,1] + -1.268;
   1:L PR[91] R[100]mm/sec CNT100 TB   .50sec,CALL END_PUD;
   1:  DO[117:Laser Start]=OFF;
   1:  PR[92] = PR[91];
   1:  PR[92,3] = PR[92,3] + 50;
   1:J PR[92] 10% FINE;
   1:  WAIT   5.00(sec);
   1:  DO[119:Gas]=OFF;
   1:  CALL HOME_ALL;
/POS
/END
